FUNCTION_BLOCK TextWriter IMPLEMENTS ITF_Writer
VAR
END_VAR

METHOD WriteMessage : BOOL
VAR_INPUT
	SomeString	: STRING(80);
END_VAR
ADSLOGSTR(msgCtrlMask := ADSLOG_MSGTYPE_LOG, msgFmtStr := 'I wrote a Text line with: %s',strArg := SomeString);
END_METHOD

END_FUNCTION_BLOCK

(* stored: Version 1.1.0.1, ProductVersion 3.1.4024.12
   POU TextWriter: Id {bdb4051e-841a-46c1-94bf-6ccad23ae39e}, SpecialFunc None
   Method WriteMessage: Id {e29b27ff-18ba-4363-9bb1-c18379a5f128} *)
